{attribute addProperty BoxType "EL2819-0000-0016"}
{attribute addProperty Id "ChannelAT %I*ARRAY[0 ..15] OF Channel_38C6D80F6480"}
{attribute addProperty CRC "3650423173"}
{attribute addProperty SizeInBites "64"}
{attribute addProperty SizeInBytes "8"}
TYPE DIG_Diag_Inputs_2815A255 :
STRUCT
	{attribute addProperty Name "Channel"}
	Channel AT %I* : ARRAY[0 ..15] OF Channel_38C6D80F;
END_STRUCT
END_TYPE

(* stored: Version 1.2.0.0, ProductVersion 3.1.4024.9
   DUT DIG_Diag_Inputs_2815A255: Id {40e6f8a3-179e-47ae-8cf7-85c170e7360c} *)
